FUNCTION_BLOCK Sensor IMPLEMENTS I_Sensor
VAR
	_name : T_MAXSTRING;
END_VAR

METHOD PUBLIC Accept
VAR_INPUT
	Visitor : I_VisitSensors;
END_VAR
Visitor.VisitSensor(this^);
END_METHOD

METHOD FB_init : BOOL
VAR_INPUT
	bInitRetains : BOOL; // if TRUE, the retain variables are initialized (warm start / cold start)
	bInCopyCode : BOOL;  // if TRUE, the instance afterwards gets moved into the copy code (online change)
	Name : T_MAXSTRING;
END_VAR
_name := Name;
END_METHOD

PROPERTY PUBLIC Name : T_MAXSTRING
GET
Name := _name;
END_GET
END_PROPERTY

END_FUNCTION_BLOCK

(* stored: Version 1.1.0.1, ProductVersion 3.1.4024.12
   POU Sensor: Id {118f2f9f-f8f3-401f-a74c-0f78b157dec5}, SpecialFunc None
   Folder Constructor: Id {e25e5da8-c123-42c0-9704-dcf6c5a87ea9}
   Method Accept: Id {da742491-9fc7-4d2c-bab3-9f10402972b4}
   Method FB_init: Id {1ac5f73f-703b-44b3-9de5-81b20067047b}
   Property Name: Id {b204250e-a703-43d3-8e82-25a9a443ce81}
   Get Get: Id {ae6ac7e8-f99f-4995-b6e5-e6cbd6cf1986} *)
